DATA_BLOCK "dbArchiveAutoTank"
{ S7_Optimized_Access := 'TRUE' }
VERSION : 0.8
NON_RETAIN
"fbArchiveAutoTank"

BEGIN

END_DATA_BLOCK

